SUBAPPLICATION DDS_PUB (* Wrapper for DDS Publisher *)
  (* Standard: 61499-2 *)
  (* Version 1.0, 2023-03-15, Tim Hesse *)
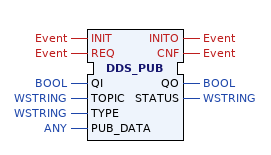
  EVENT_INPUT
    INIT; (* Initialization Request *)
    REQ; (* Normal Execution Request *)
  END_EVENT
  EVENT_OUTPUT
    INITO; (* Initialization Confirm *)
    CNF; (* Execution Confirmation *)
  END_EVENT
  VAR_INPUT
    QI : BOOL; (* Input event qualifier *)
    TOPIC : WSTRING; (* DDS Topic *)
    TYPE : WSTRING; (* DDS Type *)
    PUB_DATA : ANY; (* Data to publish *)
  END_VAR
  VAR_OUTPUT
    QO : BOOL; (* Output event qualifier *)
    STATUS : WSTRING; (* Service Status *)
  END_VAR
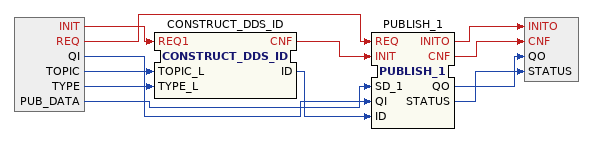
  FBS
    PUBLISH_1 : PUBLISH_1;
    CONSTRUCT_DDS_ID : CONSTRUCT_DDS_ID;
  END_FBS
  EVENT_CONNECTIONS
    PUBLISH_1.INITO TO INITO;
    PUBLISH_1.CNF TO CNF;
    REQ TO PUBLISH_1.REQ;
    INIT TO CONSTRUCT_DDS_ID.REQ1;
    CONSTRUCT_DDS_ID.CNF TO PUBLISH_1.INIT;
  END_CONNECTIONS
  DATA_CONNECTIONS
    PUB_DATA TO PUBLISH_1.SD_1;
    QI TO PUBLISH_1.QI;
    PUBLISH_1.QO TO QO;
    PUBLISH_1.STATUS TO STATUS;
    TOPIC TO CONSTRUCT_DDS_ID.TOPIC_L;
    TYPE TO CONSTRUCT_DDS_ID.TYPE_L;
    CONSTRUCT_DDS_ID.ID TO PUBLISH_1.ID;
  END_CONNECTIONS
END_SUBAPPLICATION
